{attribute 'GeneratedUsingTerminal: EL6224-0000-0021'}
{attribute addProperty BoxType "EL6224-0000-0021"}
{attribute addProperty Id "Bitheader_1AT %I*BYTE1Byte_xAT %I*ARRAY[0..7] OF BYTE8Bitheader_2AT %I*BYTE1"}
{attribute addProperty CRC "50343685"}
{attribute addProperty Size "10"}
TYPE IO_Link_Port1_in_4EEDF10D EXTENDS InputBase_8311D824 :
STRUCT
	{attribute addProperty Name "Bitheader_1"}
	Bitheader_1 AT %I* : BYTE;
	{attribute addProperty Name "Byte"}
	Byte_x AT %I* : ARRAY[0..7] OF BYTE;
	{attribute addProperty Name "Bitheader_2"}
	Bitheader_2 AT %I* : BYTE;
END_STRUCT
END_TYPE

(* stored: Version 1.2.0.0, ProductVersion 3.1.4024.11
   DUT IO_Link_Port1_in_4EEDF10D: Id {49526595-0a81-4fd6-8d65-31fa896036ca} *)
